TYPE E_ReturnMode : (
    RETURN_MODE_LOCAL := 0,
    RETURN_MODE_REFERENCE := 10
); END_TYPE

(* stored: Version 1.1.0.1
   DUT E_ReturnMode: Id {E3000000-0000-4000-8000-000000000019} *)
